// TwinCAT 3 PLC project MyFirstVersionControlled
// ProgramVersion: 3.1.4023.0
// libraries:
//   Tc2_Standard, * (Beckhoff Automation GmbH)
//   Tc2_System, * (Beckhoff Automation GmbH)
//   Tc3_Module, * (Beckhoff Automation GmbH)
// project tree:
//   / PlcTask.TcTTO
//   POUs/ FB_Alarms.TcPOU, FB_CommandAndControl.TcPOU, FB_Counter.TcPOU, MAIN.TcPOU
// real-time tasks:
//   TASK PlcTask: cycle T#10ms, priority 20, ADS port 350
//   TASK PlcTask1: cycle T#10ms, priority 21, ADS port 351

CONFIGURATION MyFirstVersionControlled
    RESOURCE PLC ON TwinCAT3
        TASK PlcTask(INTERVAL := T#10ms, PRIORITY := 21);
        PROGRAM MAIN WITH PlcTask : MAIN;
    END_RESOURCE
END_CONFIGURATION

// ---- POUs/MAIN.TcPOU
PROGRAM MAIN
VAR
	fbCounter : FB_Counter;
	fbCounter2 : FB_Counter;
	
END_VAR

fbCounter.M_AddCounterValue();

fbCounter2.M_AddCounterValue();

END_PROGRAM

// ---- POUs/FB_Counter.TcPOU
FUNCTION_BLOCK FB_Counter

VAR
	vdiCounterValue : DINT;
END_VAR

METHOD M_AddCounterValue
VAR
END_VAR
vdiCounterValue := vdiCounterValue + 1;
END_METHOD

END_FUNCTION_BLOCK

// ---- POUs/FB_Alarms.TcPOU
FUNCTION_BLOCK FB_Alarms
VAR_INPUT
END_VAR
VAR_OUTPUT
END_VAR
VAR
END_VAR

METHOD M_IntializeAlarms
VAR_INPUT
END_VAR
END_METHOD

END_FUNCTION_BLOCK

// ---- POUs/FB_CommandAndControl.TcPOU
FUNCTION_BLOCK FB_CommandAndControl
VAR_INPUT
END_VAR
VAR_OUTPUT
END_VAR
VAR
END_VAR

METHOD M_InitializeCounter
VAR_INPUT
END_VAR
END_METHOD

END_FUNCTION_BLOCK
